// TIA Portal V21 export
VAR_GLOBAL   // PLC tag table "KAllComun"
END_VAR
VAR_GLOBAL CONSTANT   // user constants
   KAllComun_PUT_Alarm : Int := 1;
   KAllComun_Get_Alarm : Int := 2;
   KAllComun_Watchdog : Int := 5;
END_VAR
